PROGRAM MAIN
VAR
	{attribute 'foobar' := 'helloworld'}
	myBool : BOOL;
	
	found : BOOL;	
	attributeValue : STRING(80);
END_VAR

found := TryReadAttributeValue('Main.myBool','foobar', adr(attributeValue), sizeof(attributeValue));

END_PROGRAM

(* stored: Version 1.1.0.1, ProductVersion 3.1.4024.12
   POU MAIN: Id {80cff89d-4624-4752-9e14-33a99f1b6cd6}, SpecialFunc None *)
